FUNCTION_BLOCK E_DEMUX_ColorMatch (* Event demultiplexor *)
  (* Standard: 61499-1 Annex A; Description: Copyright (c) 2017 fortiss GmbH This program and the accompanying materials are made available under the terms of the Eclipse Public License 2.0 which is available at https://www.eclipse.org/legal/epl-2.0/ SPDX-License-Identifier: EPL-2.0 *)
  (* Version 1.0, 2017-09-22, Alois Zoitl, fortiss GmbH, initial API and implementation and/or initial documentation *)
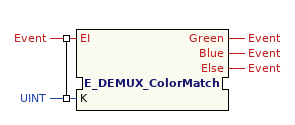
  EVENT_INPUT
    EI WITH K;
  END_EVENT
  EVENT_OUTPUT
    Green;
    Blue;
    Else;
  END_EVENT
  VAR_INPUT
    K : UINT;
  END_VAR
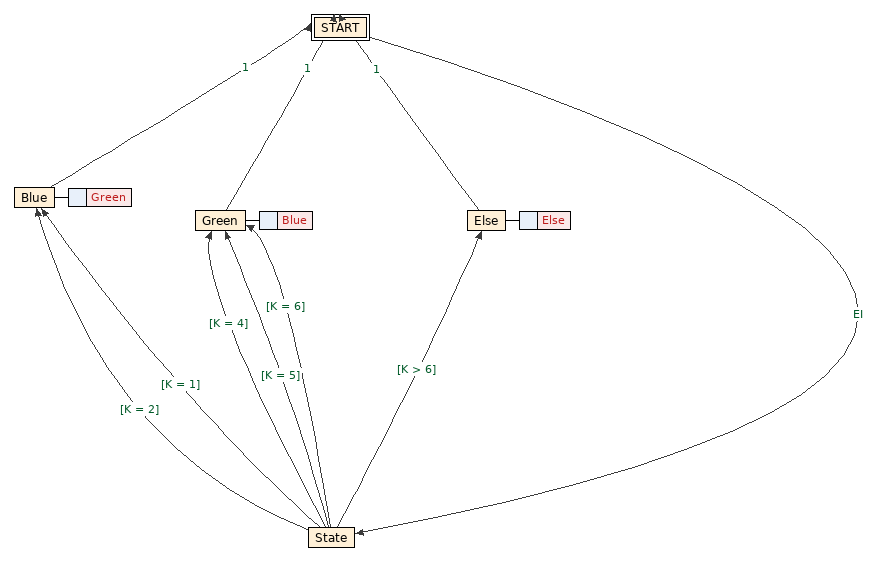
  EC_STATES
    START; (* Initial State *)
    State;
    Blue : -> Green;
    Green : -> Blue;
    Else : -> Else;
  END_STATES
  EC_TRANSITIONS
    Blue TO START := 1;
    Green TO START := 1;
    Else TO START := 1;
    START TO State := EI;
    State TO Blue := [K = 1];
    State TO Green := [K = 4];
    State TO Else := [K > 6];
    State TO Blue := [K = 2];
    State TO Green := [K = 5];
    State TO Green := [K = 6];
  END_TRANSITIONS
END_FUNCTION_BLOCK
